FUNCTION_BLOCK E_DEMUX
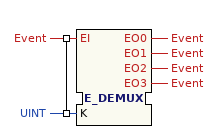
  EVENT_INPUT
    EI WITH K;
  END_EVENT
  EVENT_OUTPUT
    EO0;
    EO1;
    EO2;
    EO3;
  END_EVENT
  VAR_INPUT
    K : UINT;
  END_VAR
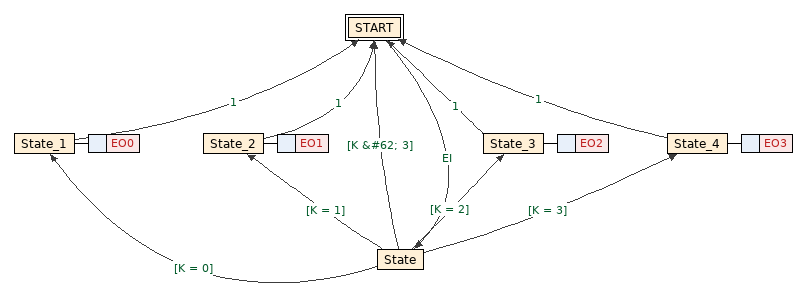
  EC_STATES
    START;
    State;
    State_1 : -> EO0;
    State_2 : -> EO1;
    State_3 : -> EO2;
    State_4 : -> EO3;
  END_STATES
  EC_TRANSITIONS
    State_1 TO START := 1;
    State_2 TO START := 1;
    State_3 TO START := 1;
    State_4 TO START := 1;
    START TO State := EI;
    State TO State_1 := [K = 0];
    State TO State_2 := [K = 1];
    State TO State_3 := [K = 2];
    State TO State_4 := [K = 3];
    State TO START := [K &#62; 3];
  END_TRANSITIONS
END_FUNCTION_BLOCK
